// TIA Portal V19 export
ORGANIZATION_BLOCK "Rack or station failure"   // OB86, LAD, RackOrStationFailure
{ S7_Optimized_Access := 'TRUE' }
// stored: SetENOAutomatically false
   VAR_INPUT
      LADDR : HW_DEVICE;   // Hardware identifier
      Event_Class : Byte;   // Event class
      Fault_ID : Byte;   // Fault identifier
   END_VAR
BEGIN
END_ORGANIZATION_BLOCK
